TYPE ST_HmiAxisSet :
STRUCT
    fRelDistance : LREAL := 60.0;   // HMI 写入：相对运动距离
    fAbsPosition : LREAL := 0.0;    // HMI 写入：绝对运动目标位置
END_STRUCT
END_TYPE

(* stored: Version 1.1.0.1, ProductVersion 3.1.4026.18
   DUT ST_HmiAxisSet: Id {7c64afe3-074a-4d9f-a713-8053332c9c55} *)
